// TIA Portal project "lab3" (V15)

(* hardware
DEVICE "S7-1200 station_1"  S7-1200 Station
   slot 0: "Rack_0"  S7-1200 Rack  Rack  V1.0
   slot 1: "PLC_1"  CPU 1214C DC/DC/DC  6ES7 214-1AG40-0XB0  V4.2
      slot 3: "AQ 1x12BIT_1"  AQ1 signal board  6ES7 232-4HA30-0XB0  V1.0
   slot 101: "CM 1243-5"  CM 1243-5  6GK7 243-5DX30-0XE0  V1.3
   slot 102: "CM 1241 (RS485)_1"  CM 1241 (RS485)  6ES7 241-1CH30-0XB0  V1.0
*)

// ===== PLC "PLC_1"  CPU 1214C DC/DC/DC =====

VAR_GLOBAL   // PLC tag table "Default tag table"
   "StartStop" AT %I0.0 : Bool;
   "zwrot" AT %M10.0 : Bool;
   "podzielnik" AT %Q0.0 : Bool;
   "CLewo" AT %I0.2 : Bool;
   "CPrawo" AT %I0.3 : Bool;
   "kLewo" AT %Q0.1 : Bool;
   "kPrawo" AT %Q0.2 : Bool;
   "zbocze1" AT %M10.1 : Bool;
   "zbocze2" AT %M10.2 : Bool;
   "zbocze3" AT %M10.3 : Bool;
   "krotki" AT %I0.4 : Bool;
   "CKrotki" AT %M11.0 : Bool;
   "sredni" AT %I0.5 : Bool;
   "dlugi" AT %I0.6 : Bool;
   "CzDlugi" AT %M11.2 : Bool;
   "zboczeKrotka" AT %M12.0 : Bool;
   "zboczeSrednia" AT %M12.1 : Bool;
   "CSredni" AT %M11.1 : Bool;
   "zboczeDluga" AT %M12.2 : Bool;
   "wyjscie_krotki" AT %Q0.4 : Bool;
   "wyjscie_sredni" AT %Q0.5 : Bool;
   "wyjscie_dlugi" AT %Q0.6 : Bool;
END_VAR

ORGANIZATION_BLOCK "Main"   // OB1, LAD, ProgramCycle
TITLE = "Main Program Sweep (Cycle)"
{ S7_Optimized_Access := 'TRUE' }
VERSION : 0.1
   VAR_INPUT
      Initial_Call : Bool;   // Initial call of this OB
      Remanence : Bool;   // =True, if remanent data are available
   END_VAR
   VAR_TEMP   // added for the SCL form of the ladder/FBD networks
      _w1 : Bool;
   END_VAR
BEGIN

REGION Network 1: podzielnik binarny
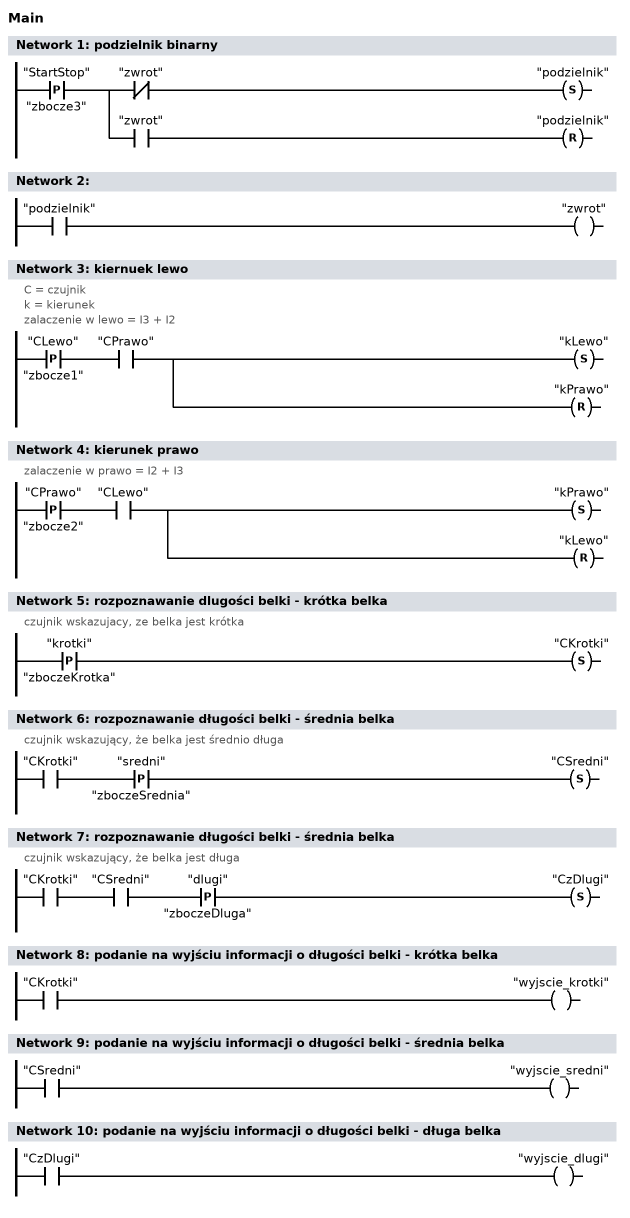
   RUNG wire#powerrail
      P_Contact(operand := "StartStop", bit := "zbocze3")
      wire#w1
      I_Contact( "zwrot" )
      S_Coil( "podzielnik" )
   END_RUNG
   RUNG wire#w1
      Contact( "zwrot" )
      R_Coil( "podzielnik" )
   END_RUNG
   // the same network as SCL:
   #_w1 := "StartStop" AND NOT "zbocze3";   // rising edge of "StartStop"
   "zbocze3" := "StartStop";
   IF #_w1 AND NOT "zwrot" THEN "podzielnik" := TRUE; END_IF;
   IF #_w1 AND "zwrot" THEN "podzielnik" := FALSE; END_IF;
END_REGION

REGION Network 2
   RUNG wire#powerrail
      Contact( "podzielnik" )
      Coil( "zwrot" )
   END_RUNG
   // the same network as SCL:
   "zwrot" := "podzielnik";
END_REGION

REGION Network 3: kiernuek lewo
   // C = czujnik
   // k = kierunek
   // zalaczenie w lewo = I3 + I2
   RUNG wire#powerrail
      P_Contact(operand := "CLewo", bit := "zbocze1")
      Contact( "CPrawo" )
      wire#w1
      S_Coil( "kLewo" )
   END_RUNG
   RUNG wire#w1
      R_Coil( "kPrawo" )
   END_RUNG
   // the same network as SCL:
   #_w1 := "CLewo" AND NOT "zbocze1";   // rising edge of "CLewo"
   "zbocze1" := "CLewo";
   IF #_w1 AND "CPrawo" THEN
       "kLewo" := TRUE;
       "kPrawo" := FALSE;
   END_IF;
END_REGION

REGION Network 4: kierunek prawo
   // zalaczenie w prawo = I2 + I3
   RUNG wire#powerrail
      P_Contact(operand := "CPrawo", bit := "zbocze2")
      Contact( "CLewo" )
      wire#w1
      S_Coil( "kPrawo" )
   END_RUNG
   RUNG wire#w1
      R_Coil( "kLewo" )
   END_RUNG
   // the same network as SCL:
   #_w1 := "CPrawo" AND NOT "zbocze2";   // rising edge of "CPrawo"
   "zbocze2" := "CPrawo";
   IF #_w1 AND "CLewo" THEN
       "kPrawo" := TRUE;
       "kLewo" := FALSE;
   END_IF;
END_REGION

REGION Network 5: rozpoznawanie dlugości belki - krótka belka
   // czujnik wskazujacy, ze belka jest krótka
   RUNG wire#powerrail
      P_Contact(operand := "krotki", bit := "zboczeKrotka")
      S_Coil( "CKrotki" )
   END_RUNG
   // the same network as SCL:
   #_w1 := "krotki" AND NOT "zboczeKrotka";   // rising edge of "krotki"
   "zboczeKrotka" := "krotki";
   IF #_w1 THEN "CKrotki" := TRUE; END_IF;
END_REGION

REGION Network 6: rozpoznawanie długości belki - średnia belka
   // czujnik wskazujący, że belka jest średnio długa
   RUNG wire#powerrail
      Contact( "CKrotki" )
      P_Contact(operand := "sredni", bit := "zboczeSrednia")
      S_Coil( "CSredni" )
   END_RUNG
   // the same network as SCL:
   #_w1 := "CKrotki" AND "sredni" AND NOT "zboczeSrednia";   // rising edge of "sredni"
   "zboczeSrednia" := "sredni";
   IF #_w1 THEN "CSredni" := TRUE; END_IF;
END_REGION

REGION Network 7: rozpoznawanie długości belki - średnia belka
   // czujnik wskazujący, że belka jest długa
   RUNG wire#powerrail
      Contact( "CKrotki" )
      Contact( "CSredni" )
      P_Contact(operand := "dlugi", bit := "zboczeDluga")
      S_Coil( "CzDlugi" )
   END_RUNG
   // the same network as SCL:
   #_w1 := "CKrotki" AND "CSredni" AND "dlugi" AND NOT "zboczeDluga";   // rising edge of "dlugi"
   "zboczeDluga" := "dlugi";
   IF #_w1 THEN "CzDlugi" := TRUE; END_IF;
END_REGION

REGION Network 8: podanie na wyjściu informacji o długości belki - krótka belka
   RUNG wire#powerrail
      Contact( "CKrotki" )
      Coil( "wyjscie_krotki" )
   END_RUNG
   // the same network as SCL:
   "wyjscie_krotki" := "CKrotki";
END_REGION

REGION Network 9: podanie na wyjściu informacji o długości belki - średnia belka
   RUNG wire#powerrail
      Contact( "CSredni" )
      Coil( "wyjscie_sredni" )
   END_RUNG
   // the same network as SCL:
   "wyjscie_sredni" := "CSredni";
END_REGION

REGION Network 10: podanie na wyjściu informacji o długości belki - długa belka
   RUNG wire#powerrail
      Contact( "CzDlugi" )
      Coil( "wyjscie_dlugi" )
   END_RUNG
   // the same network as SCL:
   "wyjscie_dlugi" := "CzDlugi";
END_REGION
END_ORGANIZATION_BLOCK